{attribute 'qualified_only'}
// Robot8 --joints parameters of setup arms
VAR_GLOBAL
	// absolute encoder value at minimal joint positon
	g_minLinkEncoder :ARRAY[1..g_sArmNum, 1..g_setupJntNum] OF DINT :=
		[123569, 35609025, 57736, 7242080, 8849999,
		 76588 , 33880077, 23270, 11506200, 2528900,
		  92809, 39087738, 30100, 90344, 45244,
		  97353, 37341559, 26764, 2969850, 13989400];
		 
	// absolute encoder value at maximum joint positon
	g_maxLinkEncoder :ARRAY[1..g_sArmNum, 1..g_setupJntNum] OF DINT :=
		[29697 , 34190666, 1678, 5374722, 468900,
		 113660, 32457000, 31924, 9643400, 10948070,
		 129919 , 37687900,  39566, 104908, 111011,
		  4419 , 35927748, 36194, 1105500, 5653000];
	
	// absolute encoder value at calibrated positon
	g_caliLinkEncoder :ARRAY[1..g_sArmNum, 1..g_setupJntNum] OF DINT :=
		[10043, 34190666, 57736, 14420666, 13062300,
		  94700, 32457000, 23270, 1922210, 6757000,
		 111618, 37687900, 30100 , 35294, 78076,
		  117777, 35927748, 26764, 10044500, 1409000];
	
	 // if absolute encoder value cross zeros within joint motion range
	g_linkEncZeroCross :ARRAY[1..g_sArmNum, 1..g_setupJntNum] OF INT :=
		[1, 0, 1, 1, 1,
		 0, 0, 0, 1, 0,
		 0, 0, 0, 1, 0,
		 1, 0, 0, 1, 1];
		 
//################ DO NOT modify parameters below ###########################
	// abolute encoder expanded limit buffer in case there is calibrtion error at limit position
    g_linkEncLimitBuffer : ARRAY [1..g_setupJntNum] OF DINT := [2000, 100000, 100, 2(100000)];
	g_linkEncLimitBufferFR : ARRAY [1..g_setupJntNum] OF DINT := [2(2000),100, 2(2000)];

	// absolute encoder direction
	g_asbEncoderDir :ARRAY[1..g_setupJntNum] OF INT :=[1, -1, 1, 1, -1];
	g_asbEncoderDirFR :ARRAY[1..g_setupJntNum] OF INT :=[1, -1, 1, -1, 1];
													
	// flag if joint can rotate multiple cycles
	g_multipleCyclesJoint :ARRAY[1..g_sArmNum, 1..g_setupJntNum] OF INT :=
		[0, 0, 0, 0, 0,
		 0, 0, 0, 0, 0,
		 0, 0, 0, 0, 0,
		 0, 0, 0, 0, 0];
		 
	// joint position at link encoder calibrated point
	g_linkEncCaliJntPos :ARRAY[1..g_sArmNum, 1..g_setupJntNum] OF LREAL :=
		[-140*g_deg2Rad, 0.779, 0.0, 90.0*g_deg2Rad, 0.0,
		 -115*g_deg2Rad, 0.607, 0.0, 90.0*g_deg2Rad, 0.0,
		 -65*g_deg2Rad, 0.607, 0.0, 90.0*g_deg2Rad, 0.0,
 		 -40*g_deg2Rad, 0.779, 0.0, 90.0*g_deg2Rad, 0.0];
	
END_VAR

(* stored: Version 1.1.0.1, ProductVersion 3.1.4024.11
   GVL GVL_SetupJointEncoderCaliData: Id {5517e73b-b8e6-4762-9cce-ad4bc8f947d8} *)
